// TIA Portal V17 program export: 1 tag tables, 1 data types, 0 data blocks, 2 code blocks (in call order from the OBs), 1 instance data blocks

VAR_GLOBAL   // PLC tag table "Convoyeur"
   Start_Button AT %I0.0 : Bool;   // Bouton marche
   Stop_Button AT %I0.1 : Bool;
   Lamp AT %Q0.0 : Bool;
   Speed_Display AT %MD20 : Real;   //    {ExternalWritable false}
END_VAR
VAR_GLOBAL CONSTANT   // user constants
   MaxStarts : Int := 1000;
END_VAR

TYPE "Recipe"
   STRUCT
      "Name" : String[20] := 'Standard';
      Speed : Real := 1.5;
      Limits : Struct
         Min : Int;
         Max : Int := 100;
      END_STRUCT;
   END_STRUCT;
END_TYPE

ORGANIZATION_BLOCK "Main"   // OB1, SCL, ProgramCycle
   VAR_INPUT
      Initial_Call : Bool;
      Remanence : Bool;
   END_VAR
   VAR_TEMP
      speed : Real;
   END_VAR
BEGIN
   "Conveyor_DB"(Start := "Start_Button", Stop := "Stop_Button");
   // vitesse en tr/min
   #speed := INT_TO_REAL(in := "Conveyor_DB".Count) * 2.5;
   IF %M10.1 THEN
       "Speed_Display" := #speed;
   END_IF;
END_ORGANIZATION_BLOCK

FUNCTION_BLOCK "Conveyor"   // FB3, LAD
{ S7_Optimized_Access := 'TRUE' }
// Convoyeur avec démarrage temporisé
   VAR_INPUT
      Start : Bool;
      Stop : Bool;   // Arrêt (contact NF)
      Delay : Time := T#2S;
   END_VAR
   VAR_OUTPUT
      Running : Bool;
      Count : Int;
   END_VAR
   VAR
      StartTimer : TON_TIME;
      Starts : CTU_INT;
      StartEdge : Bool;
      Latched : Bool;
   END_VAR
   VAR_TEMP   // added for the SCL form of the ladder/FBD networks
      _w1 : Bool;
   END_VAR
BEGIN

REGION Network 1: Auto-maintien
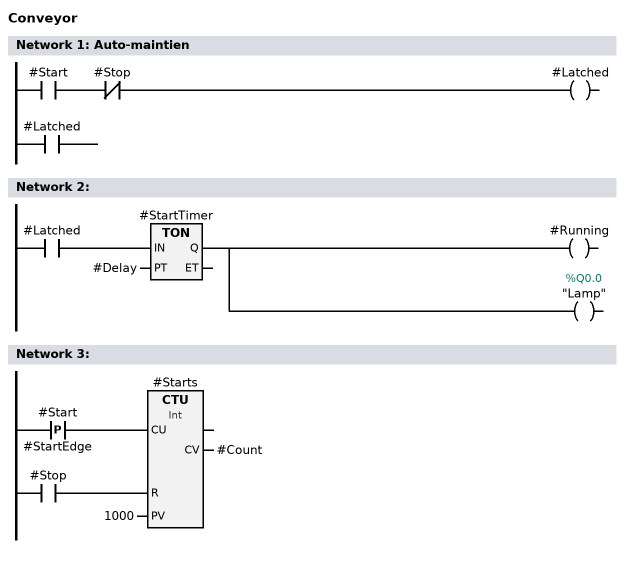
   #Latched := #Start AND NOT #Stop;
END_REGION

REGION Network 2
   RUNG wire#powerrail
      Contact( #Latched )
      #StartTimer.TON(pt := #Delay, et =>)
      wire#w1
      Coil( #Running )
   END_RUNG
   RUNG wire#w1
      Coil( "Lamp" )
   END_RUNG
   // the same network as SCL:
   #StartTimer(IN := #Latched, PT := #Delay);   // TON
   #Running := #StartTimer.Q;
   "Lamp" := #StartTimer.Q;
END_REGION

REGION Network 3
   #_w1 := #Start AND NOT #StartEdge;   // rising edge of #Start
   #StartEdge := #Start;
   #Starts(CU := #_w1, R := #Stop, PV := 1000, CV => #Count);   // CTU
END_REGION
END_FUNCTION_BLOCK

DATA_BLOCK "Conveyor_DB"   // DB3
// stored: InstanceOfName Conveyor, InstanceOfType FB
"Conveyor"
BEGIN
END_DATA_BLOCK
